Staubli VAL3: printNum.pgx

public program printNum(num& x_nInput[])
  local num l_nElement
  local num l_nLength
begin

  l_nLength = size(x_nInput)

  for l_nElement = 0 to l_nLength-1
    ? x_nInput[l_nElement]
  endFor

end
